(* PLC project OOP_Curso, Beckhoff Automation GmbH TwinCAT PLC Control 3.5.13.21 *)
(* stored: creationDateTime 2023-01-21T20:30:57.9553772, modificationDateTime 2023-01-21T20:30:57.9553772 *)

FUNCTION_BLOCK Coche
VAR_INPUT
END_VAR
VAR_OUTPUT
END_VAR
VAR
	_Marca : STRING;
	_Color : STRING;
	accion : STRING;
END_VAR

            
          

METHOD PUBLIC Acelerar
                  accion := 'acelerar';
                
END_METHOD

METHOD PUBLIC Conducir
                  accion := 'conducir';
                
END_METHOD

METHOD PUBLIC Frenar
                  accion := 'frenar';
                
END_METHOD

PROPERTY PUBLIC Color : STRING
GET
                    Color := _Color;
                  
END_GET
SET
                    _Color := Color;
                  
END_SET
END_PROPERTY

PROPERTY PUBLIC Marca : STRING
GET
                    Marca := _Marca;
                  
END_GET
SET
                    _Marca := Marca;
                  
END_SET
END_PROPERTY
END_FUNCTION_BLOCK

PROGRAM _01_Clase_y_Objetos
VAR
	// tenemos la Clase Coche y la instanciamos y obtenemos los Objetos: Mercedes, Bmw y Audi.
	Mercedes : Coche;
	Bmw : Coche;
	Audi: Coche;
	
	Color : STRING;
	Marca : STRING;
	
	Acelerar : BOOL;
	Conducir:  BOOL;
	Frenar  : BOOL;
	
	
END_VAR

            //Objeto Mercedes
//llamadas a sus métodos.
IF Acelerar THEN
	Mercedes.Acelerar();
	Acelerar := FALSE;
END_IF

IF Conducir THEN
	Mercedes.Conducir();
	Conducir := FALSE;
END_IF

IF Frenar THEN
	Mercedes.Frenar();
	Frenar := FALSE;
END_IF

//llamadas a sus propiedades.
Mercedes.Marca := 'Mercedes';
Mercedes.Color := 'Negro';
Color := Mercedes.Color;

          
END_PROGRAM
